(* CODESYS project rfid.project

Project tree, tasks and I/O mapping:
  Device : TBEN-Lx-4RFID-8DXP-CDS, Turck, order no. 6814018, version 3.5.11.20
    application Application
      libraries: RFID universal data interface, 1.0.4.0 (TURCK); Standard, * (System); VisuDialogs, * (System); HTTP Client, 1.0.1.1 (3S - Smart Software Solutions GmbH)
      task MainTask (cyclic, interval t#20ms, priority 1) calls PLC_PRG
      program PLC_PRG [ST]
      global variables GVL
      Enums/
        data type STATE
        data type FRAG
      Functions/
        function JsonMessage [ST]
      FunctionBlocks/
        function block ClearBuffers [ST]
        function block StartRead [ST]
        function block CopyBufferValues [ST]
        function block HttpSend [ST]
    LEDs : LEDs, Turck, version 1.0.0.0
        unmapped channels: APPL LED (green), APPL LED (red)
    Local_IO : Local IO, Turck, version 1.1.3.0
      UHF_extended : UHF extended, Turck, version 1.1.3.0
          settings: HF: Bypass time ( *1ms) = 100
          input  Application.GVL.input : UHF_extended_Input  // UHF extended
          output Application.GVL.output : UHF_extended_Output  // UHF extended
      _128_Byte_read : 128 Byte read, Turck, version 1.1.3.0
          input  Application.GVL.arbReadData : ARRAY[0..127] OF BYTE  // Input buffer byte
      _128_Byte_write : 128 Byte write, Turck, version 1.1.3.0
          output Application.GVL.arbWriteData : ARRAY[0..127] OF BYTE  // Output buffer byte
      HF_compact : HF compact, Turck, version 1.1.3.0
          settings: HF: Bypass time ( *1ms) = 100
          unmapped channels: HF compact, HF compact
      _128_Byte_read_1 : 128 Byte read, Turck, version 1.1.3.0
          unmapped channels: Input buffer byte
      _128_Byte_write_1 : 128 Byte write, Turck, version 1.1.3.0
          unmapped channels: Output buffer byte
      HF_compact_2 : HF compact, Turck, version 1.1.3.0
          unmapped channels: HF compact, HF compact
      _128_Byte_read_2 : 128 Byte read, Turck, version 1.1.3.0
          unmapped channels: Input buffer byte
      _128_Byte_write_2 : 128 Byte write, Turck, version 1.1.3.0
          unmapped channels: Output buffer byte
      HF_compact_3 : HF compact, Turck, version 1.1.3.0
          unmapped channels: HF compact, HF compact
      _128_Byte_read_3 : 128 Byte read, Turck, version 1.1.3.0
          unmapped channels: Input buffer byte
      _128_Byte_write_3 : 128 Byte write, Turck, version 1.1.3.0
          unmapped channels: Output buffer byte
      RFID_diagnostics : RFID diagnostics, Turck, version 1.1.3.0
          unmapped channels: RFID diagnostics
      DXP : DXP, Turck, version 1.1.3.0
          unmapped channels: DXP, DXP
      Diagnostics : Diagnostics, Turck, version 1.1.3.0
          unmapped channels: Diagnostics
      VAUX_control : VAUX control, Turck, version 1.1.3.0
          unmapped channels: VAUX control
      Module_status : Module status, Turck, version 1.1.3.0
          unmapped channels: Module status
    Ethernet : Ethernet, Turck, version 3.5.11.20
        settings: IPAddress = [192,168,1,114]; SubnetMask = [255,255,255,0]; GatewayAddress = [192,168,1,1]; MACAddress = [16#00,16#07,16#46,16#11,16#1D,16#A7]; SaveCommunicationSettings = FALSE
  TN_UHF_Q300_xxx_CDS : TN-UHF-Q300-xxx-CDS, Turck, version 3.5.11.20
    application Application
      libraries: RFID universal data interface, 1.0.4.0 (TURCK); HTTP Client, 1.0.1.1 (3S - Smart Software Solutions GmbH); Standard, * (System)
      task MainTask (cyclic, interval t#20ms, priority 1) calls PLC_PRG
      Enums/
        data type STATE
        data type FRAG
      FunctionBlocks/
        function block ClearBuffers [ST]
        function block StartRead [ST]
        function block CopyBufferValues [ST]
        function block HttpSend [ST]
      Functions/
        function JsonMessage [ST]
      global variables GVL
      program PLC_PRG [ST]
    LEDs : LEDs, Turck, version 1.0.0.0
        unmapped channels: APPL LED (green), APPL LED (red)
    Local_IO : Local IO, Turck, version 1.0.0.0
      UHF_extended : UHF extended, Turck, version 1.0.0.0
          input  Application.GVL.input : UHF_extended_Input  // UHF extended
          output Application.GVL.output : UHF_extended_Output  // UHF extended
      _128_Byte_read : 128 Byte read, Turck, version 1.0.0.0
          input  Application.GVL.arbReadData : ARRAY[0..127] OF BYTE  // Input buffer byte
      _128_Byte_write : 128 Byte write, Turck, version 1.0.0.0
          unmapped channels: Output buffer byte
      RFID_diagnostics : RFID diagnostics, Turck, version 1.0.0.0
          unmapped channels: RFID diagnostics
      DXP : DXP, Turck, version 1.0.0.0
          unmapped channels: DXP, DXP
      DXP_diagnostics : DXP diagnostics, Turck, version 1.0.0.0
          unmapped channels: DXP diagnostics
      VAUX_control : VAUX control, Turck, version 1.0.0.0
          unmapped channels: VAUX control
      Module_status : Module status, Turck, version 1.0.0.0
          unmapped channels: Module status
    Ethernet : Ethernet, Turck, version 3.5.11.20
  libraries: VisuSymbols, 3.5.10.0 (System)
  text list GlobalTextList
*)

// Device/Application/Enums/STATE
TYPE STATE :
(
	INIT,
	CLEAR,
	READ,
	READY,
	HTTP_SEND
);
END_TYPE

// Device/Application/Enums/FRAG
TYPE FRAG :
(
	COPY,
	NEXT,
	DATA
);
END_TYPE

// TN_UHF_Q300_xxx_CDS/Application/Enums/STATE
TYPE STATE :
(
	INIT,
	CLEAR,
	READ,
	READY,
	HTTP_SEND
);
END_TYPE

// TN_UHF_Q300_xxx_CDS/Application/Enums/FRAG
TYPE FRAG :
(
	COPY,
	NEXT,
	DATA
);
END_TYPE

// Device/Application/GVL
{attribute 'qualified_only'}
VAR_GLOBAL
	// TAG ids
	IDs: ARRAY[0..31] OF BYTE;
	// Data buffer for reading
	arbReadData: ARRAY[0..127] OF BYTE;
	// Data buffer for writing
	arbWriteData: ARRAY[0..127] OF BYTE;
	// Array storing tag's EPC as string
	sTagName: ARRAY[1..100] OF DWORD;
	// Array for storing EPC for every tag [EPC], [tag no.]
	arbEPC: ARRAY [0..11,1..100] OF BYTE;
	// Array for RSSI values
	arbRSSI: ARRAY[1..100] OF REAL;
	// Array for Antenna numbers
	arbAntNumber: ARRAY [1..100] OF INT;
	// Data array for storing all read RFID data
	//arbDatabank: ARRAY[0..960] OF BYTE;
	
	//arbDatabank2: ARRAY[0..16] OF Inputs_64_bytes;
	buffer:  ARRAY[0..1023] OF BYTE;
	// RFID structure input mapping
	input: ExtendedInput_t;
	// RFID structure output mapping
	output: ExtendedOutput_t;
END_VAR

// TN_UHF_Q300_xxx_CDS/Application/GVL
{attribute 'qualified_only'}
VAR_GLOBAL
	// TAG ids
	IDs: ARRAY[0..31] OF BYTE;
	// Data buffer for reading
	arbReadData: ARRAY[0..127] OF BYTE;
	// Data buffer for writing
	arbWriteData: ARRAY[0..127] OF BYTE;
	// Array storing tag's EPC as string
	sTagName: ARRAY[1..100] OF DWORD;
	// Array for storing EPC for every tag [EPC], [tag no.]
	arbEPC: ARRAY [0..11,1..100] OF BYTE;
	// Array for RSSI values
	arbRSSI: ARRAY[1..100] OF REAL;
	// Array for Antenna numbers
	arbAntNumber: ARRAY [1..100] OF INT;
	// Data array for storing all read RFID data
	//arbDatabank: ARRAY[0..960] OF BYTE;
	
	//arbDatabank2: ARRAY[0..16] OF Inputs_64_bytes;
	buffer:  ARRAY[0..1023] OF BYTE;
	// RFID structure input mapping
	input: ExtendedInput_t;
	// RFID structure output mapping
	output: ExtendedOutput_t;
END_VAR

// Device/Application/PLC_PRG
PROGRAM PLC_PRG
VAR
	NextState: STATE;
	State: STATE;
END_VAR
VAR RETAIN
	// Variable for setting the desired reading time in ms (default is 2s)
	iReadTime: UINT := 200;
END_VAR
VAR
	// used for fragmentation
	Frag: FRAG;
	// Timer for pause between reads.
	waitTimer: TON;
	// Timer if a delay is needed before any command
	tTimer: TON;
	ClearBuffers: ClearBuffers;
	StartRead: StartRead;
	message: WSTRING;
	CopyBufferValues: CopyBufferValues;
	HttpSend: HttpSend;
END_VAR

CASE State OF
	INIT:	
		waitTimer(IN:= TRUE);
		IF waitTimer.Q THEN
			waitTimer(IN:= FALSE, PT:= T#200MS);
			// Reset command when started
			gvl.output.eCommandCode := COMMAND.IDLE;
			NextState := CLEAR;
		END_IF
	CLEAR:	
		IF gvl.input.eResponseCode = RESC.IDLE THEN
			ClearBuffers();
			NextState := READ;
		END_IF
	READ:	
		StartRead();
		NextState := READY;
	READY:
		IF gvl.input.eResponseCode = RESC.INVENTORY THEN
			CopyBufferValues();
			IF CopyBufferValues.Finished THEN
				NextState := HTTP_SEND;
			END_IF
			
		ELSIF gvl.input.wErrorCode <> ERROR.NO_ERROR  THEN
			NextState := INIT;
		END_IF
	HTTP_SEND:
		IF GVL.input.uiTagCounter > 0 THEN
			HttpSend();
			IF HttpSend.MessageSent THEN
				waitTimer(PT:= T#2000MS);
				NextState := INIT;
			END_IF
		END_IF

END_CASE
	
State := NextState;

END_PROGRAM

// Device/Application/FunctionBlocks/ClearBuffers
FUNCTION_BLOCK ClearBuffers
VAR_INPUT
END_VAR
VAR_OUTPUT
END_VAR
VAR
	i: INT;
	j: INT;
END_VAR

// clear data of IDs
FOR i:= 0 TO 31 DO
	gvl.IDs[i] := 0;
END_FOR
// clear Data Buffer
FOR j := 0 TO 1023 DO
	gvl.buffer[j] := 0;
END_FOR

END_FUNCTION_BLOCK

// TN_UHF_Q300_xxx_CDS/Application/FunctionBlocks/ClearBuffers
FUNCTION_BLOCK ClearBuffers
VAR_INPUT
END_VAR
VAR_OUTPUT
END_VAR
VAR
	i: INT;
	j: INT;
END_VAR

// clear data of IDs
FOR i:= 0 TO 31 DO
	gvl.IDs[i] := 0;
END_FOR
// clear Data Buffer
FOR j := 0 TO 1023 DO
	gvl.buffer[j] := 0;
END_FOR

END_FUNCTION_BLOCK

// Device/Application/FunctionBlocks/StartRead
FUNCTION_BLOCK StartRead
VAR_INPUT
END_VAR
VAR_OUTPUT
END_VAR
VAR
END_VAR

//set the output values for read command
gvl.output.dwAddress := 1;
gvl.output.usiUHFMemoryArea := UHF_MEMORY_AREA.EPC;
gvl.output.uiTimeout:= 200;
gvl.output.eCommandCode := COMMAND.INVENTORY;

END_FUNCTION_BLOCK

// TN_UHF_Q300_xxx_CDS/Application/FunctionBlocks/StartRead
FUNCTION_BLOCK StartRead
VAR_INPUT
END_VAR
VAR_OUTPUT
END_VAR
VAR
END_VAR

//set the output values for read command
gvl.output.dwAddress := 1;
gvl.output.usiUHFMemoryArea := 1;
gvl.output.uiTimeout:= 200;
gvl.output.eCommandCode := 1;

END_FUNCTION_BLOCK

// Device/Application/FunctionBlocks/CopyBufferValues
FUNCTION_BLOCK CopyBufferValues
VAR
	i: INT;
	pump: INT;
	m: UINT;
END_VAR
VAR_OUTPUT
	Finished: BOOL;
END_VAR
VAR
	Frag: FRAG;
END_VAR

CASE Frag OF
	COPY:
		FOR i:= 0 TO 127 DO
			gvl.buffer[i+pump] := gvl.arbReadData[i];
		END_FOR
		Frag := NEXT;
		Finished := FALSE;
	NEXT:	
// Read datafragments when needed
		IF gvl.input.usiReadFragmentNo > 0 THEN
			gvl.output.usiReadFragmentNo := gvl.output.usiReadFragmentNo + 1;	
			pump := pump + 128;
			Frag := COPY;
		ELSE
			gvl.output.usiReadFragmentNo := 0;
			pump := 0;
			Frag := DATA;
		END_IF		
		Finished := FALSE;			
	DATA:	
// Put the read data to the right order (18 byte data with RSSI configured in the antenna)
		FOR m:= 0 TO GVL.input.uiTagCounter DO
			gvl.IDS[m]:= gvl.buffer[2+18*m];
		END_FOR
		Frag := COPY;
		Finished := TRUE;
END_CASE

END_FUNCTION_BLOCK

// TN_UHF_Q300_xxx_CDS/Application/FunctionBlocks/CopyBufferValues
FUNCTION_BLOCK CopyBufferValues
VAR
	i: INT;
	pump: INT;
	m: UINT;
END_VAR
VAR_OUTPUT
	Finished: BOOL;
END_VAR
VAR
	Frag: FRAG;
END_VAR

CASE Frag OF
	COPY:
		FOR i:= 0 TO 127 DO
			gvl.buffer[i+pump] := gvl.arbReadData[i];
		END_FOR
		Frag := NEXT;
		Finished := FALSE;
	NEXT:	
// Read datafragments when needed
		IF gvl.input.usiReadFragmentNo <> 0 THEN
			gvl.output.usiReadFragmentNo := gvl.output.usiReadFragmentNo + 1;	
			pump := pump + 128;
			Frag := COPY;
		ELSE
			gvl.output.usiReadFragmentNo := 0;
			pump := 0;
			Frag := DATA;
		END_IF		
		Finished := FALSE;			
	DATA:	
// Put the read data to the right order (18 byte data with RSSI configured in the antenna)
		FOR m:= 0 TO GVL.input.uiTagCounter DO
			gvl.IDS[m]:= gvl.buffer[2+18*m];
		END_FOR
		Frag := COPY;
		Finished := TRUE;
END_CASE

END_FUNCTION_BLOCK

// Device/Application/FunctionBlocks/HttpSend
FUNCTION_BLOCK HttpSend
VAR
	send: HTTP.HttpClient;
	message: WSTRING;
END_VAR
VAR_OUTPUT
	MessageSent: BOOL;
END_VAR

message:= JsonMessage();
send(
	xExecute:= NOT MessageSent,
	udiTimeOut:= 2000000,
	sURL:= '192.168.5.1/api/production/ids',
	eRequestType:= HTTP.REQUEST_TYPE.POST,
	eContentType:= HTTP.CONTENT_TYPE.APPLICATION_JSON,
	pwsPostValue:= ADR(message)
);
MessageSent:= send.xDone OR send.xError;

END_FUNCTION_BLOCK

// Device/Application/Functions/JsonMessage
FUNCTION JsonMessage : WSTRING
VAR
	stringBuilder: STRING;
	i: INT;
END_VAR

stringBuilder := CONCAT('[',BYTE_TO_STRING(gvl.IDs[0]));
i := 1;
WHILE gvl.IDs[i] <> 0 DO
	stringBuilder := CONCAT(stringBuilder,',');
	stringBuilder := CONCAT(stringBuilder,BYTE_TO_STRING(gvl.IDs[i]));
	i := i + 1;
END_WHILE
stringBuilder := CONCAT(stringBuilder,']');
JsonMessage := STRING_TO_WSTRING(stringBuilder);

END_FUNCTION

// TN_UHF_Q300_xxx_CDS/Application/Functions/JsonMessage
FUNCTION JsonMessage : WSTRING
VAR
	stringBuilder: STRING;
	i: INT;
END_VAR

stringBuilder := CONCAT('[',BYTE_TO_STRING(gvl.IDs[0]));
i := 1;
WHILE gvl.IDs[i] <> 0 DO
	stringBuilder := CONCAT(stringBuilder,',');
	stringBuilder := CONCAT(stringBuilder,BYTE_TO_STRING(gvl.IDs[i]));
	i := i + 1;
END_WHILE
stringBuilder := CONCAT(stringBuilder,']');
JsonMessage := STRING_TO_WSTRING(stringBuilder);

END_FUNCTION

// TN_UHF_Q300_xxx_CDS/Application/FunctionBlocks/HttpSend
FUNCTION_BLOCK HttpSend
VAR
	send: HTTP.HttpClient;
	message: WSTRING;
END_VAR
VAR_OUTPUT
	MessageSent: BOOL;
END_VAR

message:= JsonMessage();
send(
	xExecute:= NOT MessageSent,
	udiTimeOut:= 2000000,
	sURL:= '192.168.5.1/api/production/ids',
	eRequestType:= HTTP.REQUEST_TYPE.POST,
	eContentType:= HTTP.CONTENT_TYPE.APPLICATION_JSON,
	pwsPostValue:= ADR(message)
);
MessageSent:= send.xDone OR send.xError;

END_FUNCTION_BLOCK

// TN_UHF_Q300_xxx_CDS/Application/PLC_PRG
PROGRAM PLC_PRG
VAR
	NextState: STATE;
	State: STATE;
END_VAR
VAR RETAIN
	// Variable for setting the desired reading time in ms (default is 2s)
	iReadTime: UINT := 200;
END_VAR
VAR
	// used for fragmentation
	Frag: FRAG;
	// Timer for pause between reads.
	waitTimer: TON;
	// Timer if a delay is needed before any command
	tTimer: TON;
	ClearBuffers: ClearBuffers;
	StartRead: StartRead;
	message: WSTRING;
	CopyBufferValues: CopyBufferValues;
	HttpSend: HttpSend;
END_VAR

CASE State OF
	INIT:	
		waitTimer(IN:= TRUE);
 		IF waitTimer.Q THEN
			waitTimer(IN:= FALSE, PT:= T#200MS);
			// Reset command when started
			gvl.output.eCommandCode := 0;
			NextState := CLEAR;
		END_IF
	CLEAR:	
		IF gvl.input.eResponseCode = 0 THEN
			ClearBuffers();
			NextState := READ;
		END_IF
	READ:	
		StartRead();
		NextState := READY;
	READY:
		IF gvl.input.eResponseCode = 1 THEN
			CopyBufferValues();
			IF CopyBufferValues.Finished THEN
				NextState := HTTP_SEND;
			END_IF
			
		ELSIF gvl.input.wErrorCode > 0  THEN
			NextState := INIT;
		END_IF
	HTTP_SEND:
		IF GVL.input.uiTagCounter > 0 THEN
			HttpSend();
			IF HttpSend.MessageSent THEN
				waitTimer(PT:= T#2000MS);
				NextState := INIT;
			END_IF
		END_IF

END_CASE
	
State := NextState;

END_PROGRAM
